// TIA Portal V17 export
// export: Created 2023-12-22T15:28:35.0741161Z, ExportSetting WithDefaults, DisplayName Totally Integrated Automation Portal, DisplayVersion V17, DisplayName TIA Portal Openness, DisplayVersion V17, DisplayName TIA Portal Version Control Interface, DisplayVersion V17, DisplayName STEP 7 Professional, DisplayVersion V17, DisplayName STEP 7 Safety, DisplayVersion V17, DisplayName WinCC Advanced, DisplayVersion V17
FUNCTION_BLOCK "DRV_Flow_old"   // FB115, LAD
{ S7_Optimized_Access := 'TRUE' }
VERSION : 0.1
// stored: AutoNumber false, IsIECCheckEnabled false, IsRetainMemResEnabled false, MemoryReserve 100, SetENOAutomatically false, UDAEnableTagReadback false
   VAR_INPUT
      Start : Bool;   // Старт
      Value : Real;   // Значение
   END_VAR
   VAR RETAIN
      Mode { S7_SetPoint := 'True'} : Bool;   // 0 - импульсный, 1 - аналоговый
   END_VAR
   VAR
      Lock : Bool;   // Блокировка учёта расхода воды
      pulse : Bool;   // Пульс
      Reset_All : Bool;   // Сброс общего счётчика
      Reset_Now : Bool;   // Сброс суточного счётчика
      Reset_Last : Bool;   // Сброс последнего счётчика
      Reset_Seans : Bool;   // Сброс счёта за сеанс
      Reset_Any : Bool;   // Сброс произвольного измерения
      Save : Bool;   // Сохранить данные за сеанс
      SaveDay : Bool;   // Сохранить данные за сутки
   END_VAR
   VAR RETAIN
      Fast_Mode { S7_SetPoint := 'True'} : Bool := True;   // Режим частых импульсов
   END_VAR
   VAR
      Inverse : Bool;   // Инверсия
      pos : Array[0..7] of Bool;   // Вспомогательные переменные
      clock { S7_SetPoint := 'True'} : Real := 0.01;   // Контроль связи 1 Гц
   END_VAR
   VAR RETAIN
      Weight { S7_SetPoint := 'True'} : Real := 1.0;   // Вес импульса
   END_VAR
   VAR
      Weight_S : Real;   // Расход за секунду
   END_VAR
   VAR RETAIN
      All { S7_SetPoint := 'True'} : Real;   // Полный расход
      Any { S7_SetPoint := 'True'} : Real;   // Произвольное измерение
      Seans { S7_SetPoint := 'True'} : Real;   // Расход за сеанс работы
      Seans_Last { S7_SetPoint := 'True'} : Real;   // Расход за прошлый сеанс
      Flow_Today { S7_SetPoint := 'True'} : Real;   // Расход за текущее измерение
      Flow_LastDay { S7_SetPoint := 'True'} : Real;   // Расход за прошлое измерение
      Flow_Lock_All { S7_SetPoint := 'True'} : Real;   // Неучтённый расход
      Flow_Lock_Now { S7_SetPoint := 'True'} : Real;   // Текущий неучтенный расхрд
   END_VAR
   VAR
      Flow_S : Real;   // Расход в секунду по импульсам
      Flow_Speed : Real;   // Скорость потока л/ч
      Pulse_CNT : Real;   // Число импульсов за время измерения
      Flow_DTM : Real;   // Низкая скорость - проток в минуту
      Flow_DT : Real;   // Время между импульсами
      Flow_clock : Real;   // Не используется
      TimeControl : "Time_R";   // Время измерения
   END_VAR
   VAR RETAIN
      Day : Int;   // Текущая дата
      ADDR_Byte { S7_SetPoint := 'True'} : Int;   // Адрес входа на контроллере (Байт)
      ADDR_Bit { S7_SetPoint := 'True'} : Int;   // Адрес входа на контроллере (Бит)
   END_VAR
   VAR
      Filter { S7_SetPoint := 'True'} : "Filter";
      Time_DTL : DTL;
   END_VAR
   VAR_TEMP
      imp : Bool;
      start_x : Bool;
      m3 : Real;
   END_VAR
   VAR CONSTANT
      Minutes : Real := 60.0;
      Hour : Real := 3600.0;
   END_VAR
   // Filter.max := 100;
   VAR_TEMP   // added for the SCL form of the ladder/FBD networks
      _w1 : Bool;
      _w2 : Bool;
   END_VAR
BEGIN

REGION Network 1: Чтение сигнала
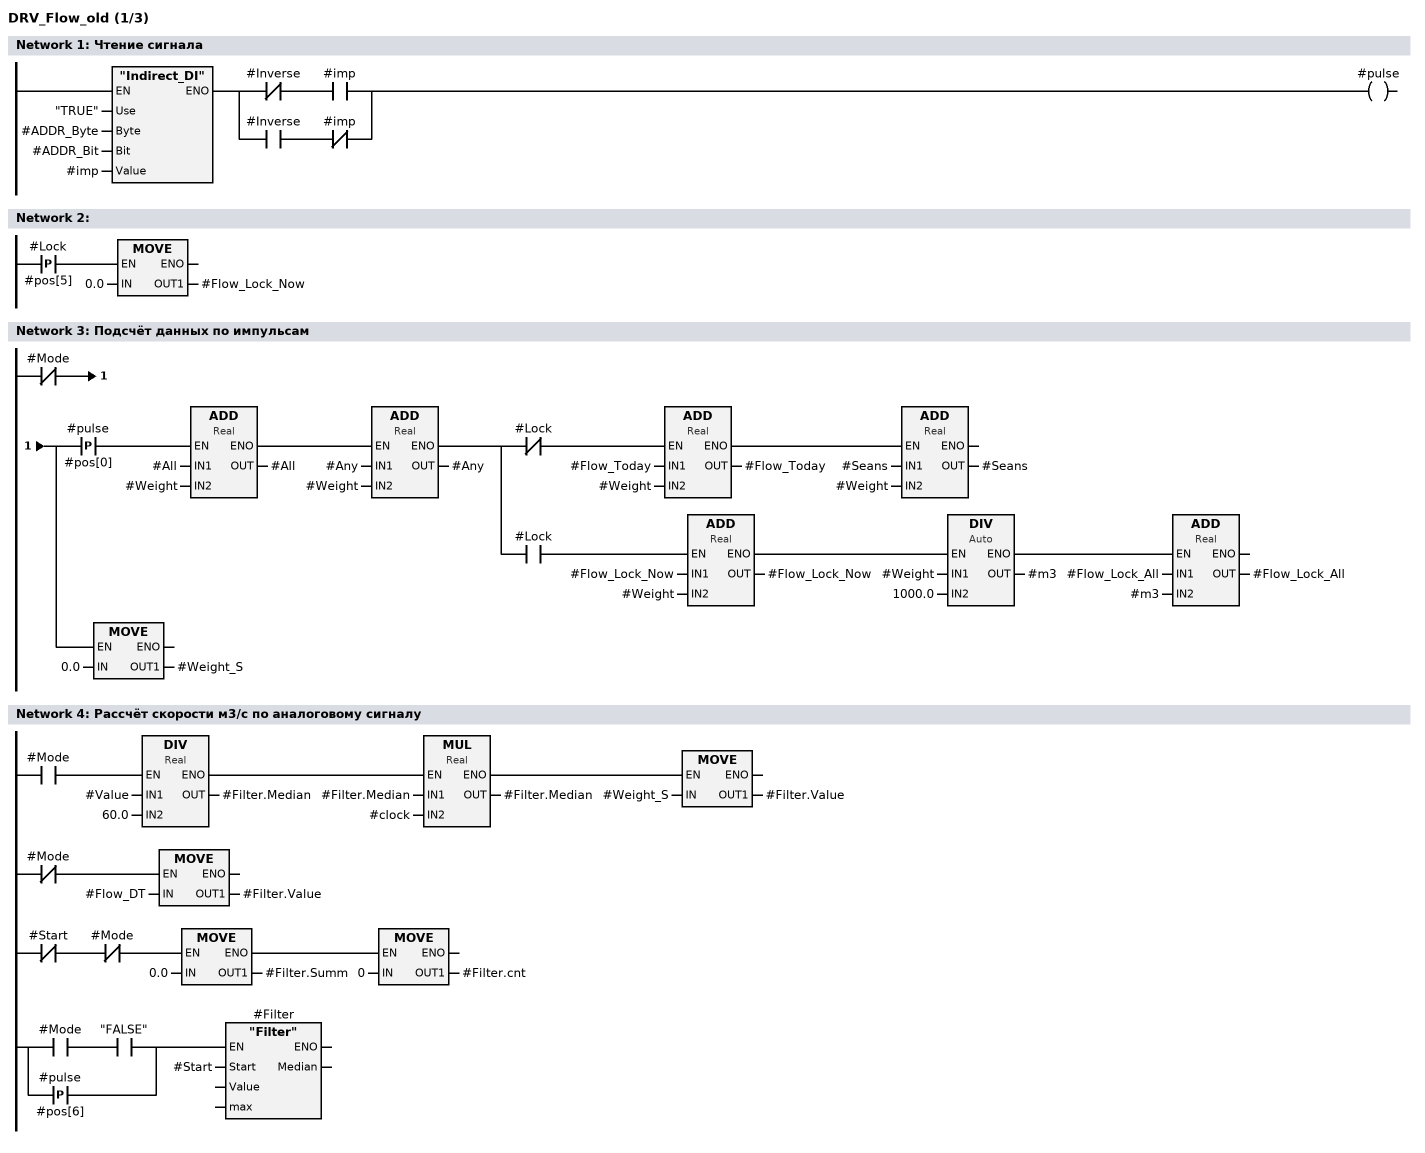
   RUNG wire#powerrail
      "Indirect_DI"(Use := "TRUE", "Byte" := #ADDR_Byte, Bit := #ADDR_Bit, Value := #imp)
      wire#w1
      I_Contact( #Inverse )
      Contact( #imp )
      wire#w2
      Coil( #pulse )
   END_RUNG
   RUNG wire#w1
      Contact( #Inverse )
      I_Contact( #imp )
   END_RUNG wire#w2
   // the same network as SCL:
   "Indirect_DI"(Use := "TRUE", "Byte" := #ADDR_Byte, Bit := #ADDR_Bit, Value := #imp, ENO => #_w1);
   #pulse := #_w1 AND ((NOT #Inverse AND #imp) OR (#Inverse AND NOT #imp));
END_REGION

REGION Network 2
   RUNG wire#powerrail
      P_Contact(operand := #Lock, bit := #pos[5])
      Move(in := 0.0, out1 => #Flow_Lock_Now)
   END_RUNG
   // the same network as SCL:
   #_w1 := #Lock AND NOT #pos[5];   // rising edge of #Lock
   #pos[5] := #Lock;
   IF #_w1 THEN #Flow_Lock_Now := 0.0; END_IF;
END_REGION

REGION Network 3: Подсчёт данных по импульсам
   RUNG wire#powerrail
      I_Contact( #Mode )
      wire#w1
      P_Contact(operand := #pulse, bit := #pos[0])
      { S7_Templates := "SrcType := Real"; S7_GenerateENO := "TRUE" } Add(in1 := #All, in2 := #Weight, out => #All)
      { S7_Templates := "SrcType := Real"; S7_GenerateENO := "TRUE" } Add(in1 := #Any, in2 := #Weight, out => #Any)
      wire#w2
      I_Contact( #Lock )
      { S7_Templates := "SrcType := Real"; S7_GenerateENO := "TRUE" } Add(in1 := #Flow_Today, in2 := #Weight, out => #Flow_Today)
      { S7_Templates := "SrcType := Real"; S7_GenerateENO := "TRUE" } Add(in1 := #Seans, in2 := #Weight, out => #Seans)
   END_RUNG
   RUNG wire#w2
      Contact( #Lock )
      { S7_Templates := "SrcType := Real"; S7_GenerateENO := "TRUE" } Add(in1 := #Flow_Lock_Now, in2 := #Weight, out => #Flow_Lock_Now)
      Div(in1 := #Weight, in2 := 1000.0, out => #m3)
      { S7_Templates := "SrcType := Real"; S7_GenerateENO := "TRUE" } Add(in1 := #Flow_Lock_All, in2 := #m3, out => #Flow_Lock_All)
   END_RUNG
   RUNG wire#w1
      Move(in := 0.0, out1 => #Weight_S)
   END_RUNG
   // the same network as SCL:
   // ENO of a box is taken as its EN; it also drops when the box reports an error
   #_w1 := NOT #Mode AND #pulse AND NOT #pos[0];   // rising edge of #pulse
   #pos[0] := #pulse;
   IF #_w1 THEN
       #All := #All + #Weight;
       #Any := #Any + #Weight;
   END_IF;
   IF #_w1 AND NOT #Lock THEN
       #Flow_Today := #Flow_Today + #Weight;
       #Seans := #Seans + #Weight;
   END_IF;
   IF #_w1 AND #Lock THEN
       #Flow_Lock_Now := #Flow_Lock_Now + #Weight;
       #m3 := #Weight / 1000.0;
       #Flow_Lock_All := #Flow_Lock_All + #m3;
   END_IF;
   IF NOT #Mode THEN #Weight_S := 0.0; END_IF;
END_REGION

REGION Network 4: Рассчёт скорости м3/с по аналоговому сигналу
   RUNG wire#powerrail
      Contact( #Mode )
      { S7_Templates := "SrcType := Real"; S7_GenerateENO := "TRUE" } Div(in1 := #Value, in2 := 60.0, out => #Filter.Median)
      { S7_Templates := "SrcType := Real"; S7_GenerateENO := "TRUE" } Mul(in1 := #Filter.Median, in2 := #clock, out => #Filter.Median)
      Move(in := #Weight_S, out1 => #Filter.Value)
   END_RUNG
   RUNG wire#powerrail
      I_Contact( #Mode )
      Move(in := #Flow_DT, out1 => #Filter.Value)
   END_RUNG
   RUNG wire#powerrail
      I_Contact( #Start )
      I_Contact( #Mode )
      Move(in := 0.0, out1 => #Filter.Summ)
      Move(in := 0, out1 => #Filter.cnt)
   END_RUNG
   RUNG wire#powerrail
      Contact( #Mode )
      Contact( "FALSE" )
      wire#w1
      #Filter(Start := #Start, Value :=, max :=, Median =>)
   END_RUNG
   RUNG wire#powerrail
      P_Contact(operand := #pulse, bit := #pos[6])
   END_RUNG wire#w1
   // the same network as SCL:
   // ENO of a box is taken as its EN; it also drops when the box reports an error
   IF #Mode THEN
       #Filter.Median := #Value / 60.0;
       #Filter.Median := #Filter.Median * #clock;
       #Filter.Value := #Weight_S;
   END_IF;
   IF NOT #Mode THEN #Filter.Value := #Flow_DT; END_IF;
   IF NOT #Start AND NOT #Mode THEN
       #Filter.Summ := 0.0;
       #Filter.cnt := 0;
   END_IF;
   #_w1 := #pulse AND NOT #pos[6];   // rising edge of #pulse
   #pos[6] := #pulse;
   IF (#Mode AND "FALSE") OR #_w1 THEN
       #Filter(Start := #Start);   // "Filter"
   END_IF;
END_REGION

REGION Network 5: Подсчёт расхода по аналоговому сигналу
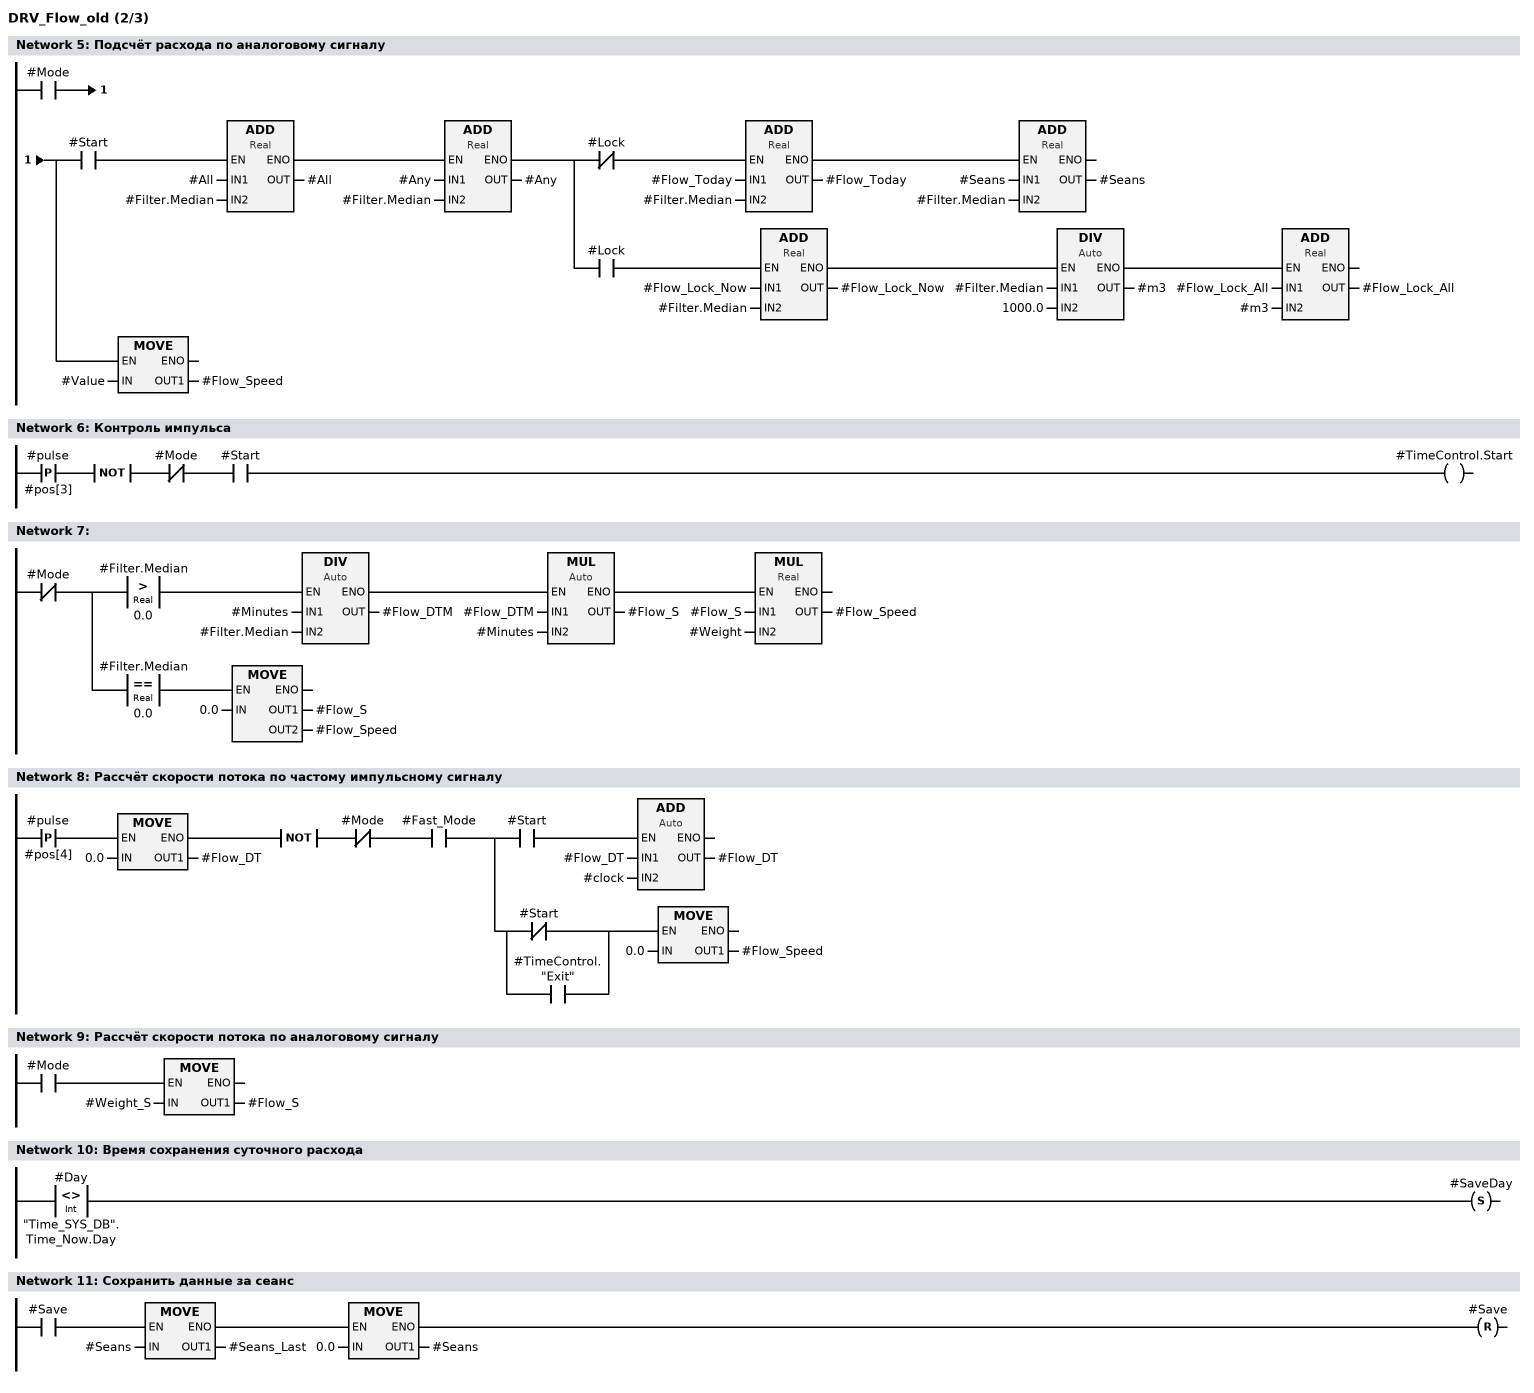
   RUNG wire#powerrail
      Contact( #Mode )
      wire#w1
      Contact( #Start )
      { S7_Templates := "SrcType := Real"; S7_GenerateENO := "TRUE" } Add(in1 := #All, in2 := #Filter.Median, out => #All)
      { S7_Templates := "SrcType := Real"; S7_GenerateENO := "TRUE" } Add(in1 := #Any, in2 := #Filter.Median, out => #Any)
      wire#w2
      I_Contact( #Lock )
      { S7_Templates := "SrcType := Real"; S7_GenerateENO := "TRUE" } Add(in1 := #Flow_Today, in2 := #Filter.Median, out => #Flow_Today)
      { S7_Templates := "SrcType := Real"; S7_GenerateENO := "TRUE" } Add(in1 := #Seans, in2 := #Filter.Median, out => #Seans)
   END_RUNG
   RUNG wire#w2
      Contact( #Lock )
      { S7_Templates := "SrcType := Real"; S7_GenerateENO := "TRUE" } Add(in1 := #Flow_Lock_Now, in2 := #Filter.Median, out => #Flow_Lock_Now)
      Div(in1 := #Filter.Median, in2 := 1000.0, out => #m3)
      { S7_Templates := "SrcType := Real"; S7_GenerateENO := "TRUE" } Add(in1 := #Flow_Lock_All, in2 := #m3, out => #Flow_Lock_All)
   END_RUNG
   RUNG wire#w1
      Move(in := #Value, out1 => #Flow_Speed)
   END_RUNG
   // the same network as SCL:
   // ENO of a box is taken as its EN; it also drops when the box reports an error
   #_w1 := #Mode AND #Start;
   IF #_w1 THEN
       #All := #All + #Filter.Median;
       #Any := #Any + #Filter.Median;
   END_IF;
   IF #_w1 AND NOT #Lock THEN
       #Flow_Today := #Flow_Today + #Filter.Median;
       #Seans := #Seans + #Filter.Median;
   END_IF;
   IF #_w1 AND #Lock THEN
       #Flow_Lock_Now := #Flow_Lock_Now + #Filter.Median;
       #m3 := #Filter.Median / 1000.0;
       #Flow_Lock_All := #Flow_Lock_All + #m3;
   END_IF;
   IF #Mode THEN #Flow_Speed := #Value; END_IF;
END_REGION

REGION Network 6: Контроль импульса
   RUNG wire#powerrail
      P_Contact(operand := #pulse, bit := #pos[3])
      Not()
      I_Contact( #Mode )
      Contact( #Start )
      Coil( #TimeControl.Start )
   END_RUNG
   // the same network as SCL:
   #_w1 := #pulse AND NOT #pos[3];   // rising edge of #pulse
   #pos[3] := #pulse;
   #TimeControl.Start := NOT #_w1 AND NOT #Mode AND #Start;
END_REGION

REGION Network 7
   RUNG wire#powerrail
      I_Contact( #Mode )
      wire#w1
      { S7_Templates := "SrcType := Real" } GT_Contact(in1 := #Filter.Median, in2 := 0.0)
      Div(in1 := #Minutes, in2 := #Filter.Median, out => #Flow_DTM)
      Mul(in1 := #Flow_DTM, in2 := #Minutes, out => #Flow_S)
      { S7_Templates := "SrcType := Real"; S7_GenerateENO := "TRUE" } Mul(in1 := #Flow_S, in2 := #Weight, out => #Flow_Speed)
   END_RUNG
   RUNG wire#w1
      { S7_Templates := "SrcType := Real" } EQ_Contact(in1 := #Filter.Median, in2 := 0.0)
      Move(in := 0.0, out1 => #Flow_S, out2 => #Flow_Speed)
   END_RUNG
   // the same network as SCL:
   IF NOT #Mode AND (#Filter.Median > 0.0) THEN
       #Flow_DTM := #Minutes / #Filter.Median;
       #Flow_S := #Flow_DTM * #Minutes;
       #Flow_Speed := #Flow_S * #Weight;
   END_IF;
   IF NOT #Mode AND (#Filter.Median = 0.0) THEN
       #Flow_S := 0.0;
       #Flow_Speed := 0.0;
   END_IF;
END_REGION

REGION Network 8: Рассчёт скорости потока по частому импульсному сигналу
   RUNG wire#powerrail
      P_Contact(operand := #pulse, bit := #pos[4])
      Move(in := 0.0, out1 => #Flow_DT)
      Not()
      I_Contact( #Mode )
      Contact( #Fast_Mode )
      wire#w1
      Contact( #Start )
      Add(in1 := #Flow_DT, in2 := #clock, out => #Flow_DT)
   END_RUNG
   RUNG wire#w1
      I_Contact( #Start )
      wire#w2
      Move(in := 0.0, out1 => #Flow_Speed)
   END_RUNG
   RUNG wire#w1
      Contact( #TimeControl."Exit" )
   END_RUNG wire#w2
   // the same network as SCL:
   #_w1 := #pulse AND NOT #pos[4];   // rising edge of #pulse
   #pos[4] := #pulse;
   IF #_w1 THEN #Flow_DT := 0.0; END_IF;
   #_w2 := NOT #_w1 AND NOT #Mode AND #Fast_Mode;
   IF #_w2 AND #Start THEN #Flow_DT := #Flow_DT + #clock; END_IF;
   IF #_w2 AND (NOT #Start OR #TimeControl."Exit") THEN #Flow_Speed := 0.0; END_IF;
END_REGION

REGION Network 9: Рассчёт скорости потока по аналоговому сигналу
   RUNG wire#powerrail
      Contact( #Mode )
      Move(in := #Weight_S, out1 => #Flow_S)
   END_RUNG
   // the same network as SCL:
   IF #Mode THEN #Flow_S := #Weight_S; END_IF;
END_REGION

REGION Network 10: Время сохранения суточного расхода
   RUNG wire#powerrail
      { S7_Templates := "SrcType := Int" } NE_Contact(in1 := #Day, in2 := "Time_SYS_DB".Time_Now.Day)
      S_Coil( #SaveDay )
   END_RUNG
   // the same network as SCL:
   IF #Day <> "Time_SYS_DB".Time_Now.Day THEN #SaveDay := TRUE; END_IF;
END_REGION

REGION Network 11: Сохранить данные за сеанс
   RUNG wire#powerrail
      Contact( #Save )
      { S7_GenerateENO := "TRUE" } Move(in := #Seans, out1 => #Seans_Last)
      { S7_GenerateENO := "TRUE" } Move(in := 0.0, out1 => #Seans)
      R_Coil( #Save )
   END_RUNG
   // the same network as SCL:
   // ENO of a box is taken as its EN; it also drops when the box reports an error
   IF #Save THEN
       #Seans_Last := #Seans;
       #Seans := 0.0;
       #Save := FALSE;
   END_IF;
END_REGION

REGION Network 12: Сохранить данные за сутки
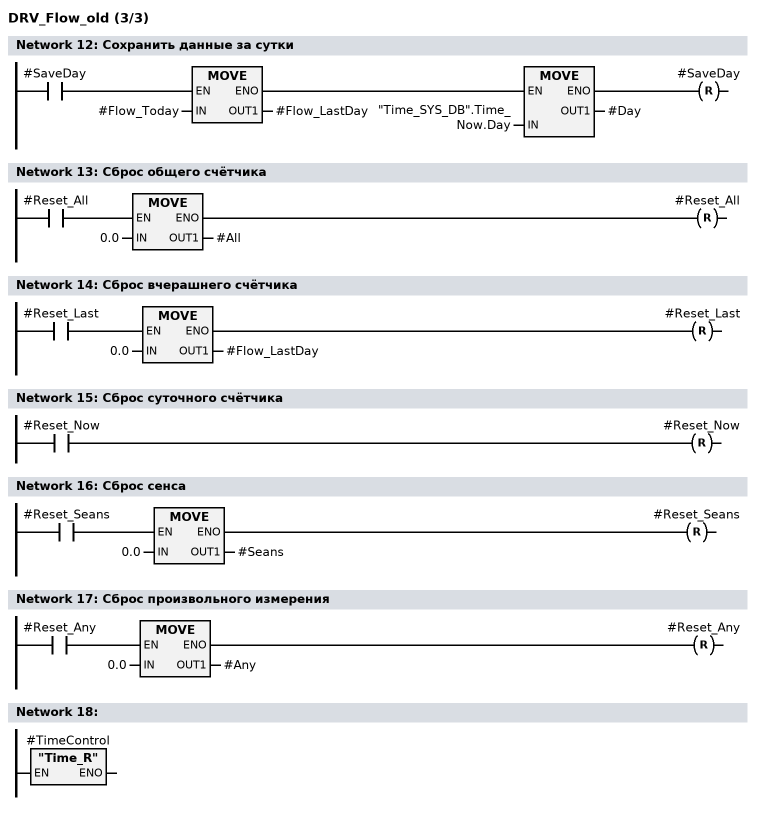
   RUNG wire#powerrail
      Contact( #SaveDay )
      { S7_GenerateENO := "TRUE" } Move(in := #Flow_Today, out1 => #Flow_LastDay)
      { S7_GenerateENO := "TRUE" } Move(in := "Time_SYS_DB".Time_Now.Day, out1 => #Day)
      R_Coil( #SaveDay )
   END_RUNG
   // the same network as SCL:
   // ENO of a box is taken as its EN; it also drops when the box reports an error
   IF #SaveDay THEN
       #Flow_LastDay := #Flow_Today;
       #Day := "Time_SYS_DB".Time_Now.Day;
       #SaveDay := FALSE;
   END_IF;
END_REGION

REGION Network 13: Сброс общего счётчика
   RUNG wire#powerrail
      Contact( #Reset_All )
      { S7_GenerateENO := "TRUE" } Move(in := 0.0, out1 => #All)
      R_Coil( #Reset_All )
   END_RUNG
   // the same network as SCL:
   // ENO of a box is taken as its EN; it also drops when the box reports an error
   IF #Reset_All THEN
       #All := 0.0;
       #Reset_All := FALSE;
   END_IF;
END_REGION

REGION Network 14: Сброс вчерашнего счётчика
   RUNG wire#powerrail
      Contact( #Reset_Last )
      { S7_GenerateENO := "TRUE" } Move(in := 0.0, out1 => #Flow_LastDay)
      R_Coil( #Reset_Last )
   END_RUNG
   // the same network as SCL:
   // ENO of a box is taken as its EN; it also drops when the box reports an error
   IF #Reset_Last THEN
       #Flow_LastDay := 0.0;
       #Reset_Last := FALSE;
   END_IF;
END_REGION

REGION Network 15: Сброс суточного счётчика
   RUNG wire#powerrail
      Contact( #Reset_Now )
      R_Coil( #Reset_Now )
   END_RUNG
   // the same network as SCL:
   IF #Reset_Now THEN #Reset_Now := FALSE; END_IF;
END_REGION

REGION Network 16: Сброс сенса
   RUNG wire#powerrail
      Contact( #Reset_Seans )
      { S7_GenerateENO := "TRUE" } Move(in := 0.0, out1 => #Seans)
      R_Coil( #Reset_Seans )
   END_RUNG
   // the same network as SCL:
   // ENO of a box is taken as its EN; it also drops when the box reports an error
   IF #Reset_Seans THEN
       #Seans := 0.0;
       #Reset_Seans := FALSE;
   END_IF;
END_REGION

REGION Network 17: Сброс произвольного измерения
   RUNG wire#powerrail
      Contact( #Reset_Any )
      { S7_GenerateENO := "TRUE" } Move(in := 0.0, out1 => #Any)
      R_Coil( #Reset_Any )
   END_RUNG
   // the same network as SCL:
   // ENO of a box is taken as its EN; it also drops when the box reports an error
   IF #Reset_Any THEN
       #Any := 0.0;
       #Reset_Any := FALSE;
   END_IF;
END_REGION

REGION Network 18
   RUNG wire#powerrail
      #TimeControl()
   END_RUNG
   // the same network as SCL:
   #TimeControl();   // "Time_R"
END_REGION
END_FUNCTION_BLOCK
